TYPE Recipe :
STRUCT
	WorkingTime: TIME; 
END_STRUCT
END_TYPE

(* stored: Version 1.1.0.1, ProductVersion 3.1.4024.12
   DUT Recipe: Id {3015f1b9-d8b7-40d5-b66f-8cb2d08060d2} *)
